INTERFACE ITF_Observer

METHOD updateConnection
VAR_INPUT
	Module : REFERENCE TO MachineModule;
END_VAR
END_METHOD

METHOD updateLock
VAR_INPUT
	setLock : BOOL;
END_VAR
END_METHOD

END_INTERFACE

(* stored: Version 1.1.0.1, ProductVersion 3.1.4024.12
   Itf ITF_Observer: Id {7fcd97c8-dddd-4c65-bfbc-c7a076a7a337}
   Method updateConnection: Id {c25919cf-b645-41c3-bb8f-6f088880249a}
   Method updateLock: Id {38e78471-25ef-429e-b095-e2cc48b34446} *)
